(* PLC project VisuTest.project, CODESYS CODESYS V3.5 SP17 Patch 2 *)
(* stored: creationDateTime 2022-02-17T09:26:16.669529, modificationDateTime 2022-02-16T16:05:59.7420926, externalized true, stored C:\development\github\xml2ooxml\out\ex_contentHeader_12.xml *)

TYPE DUT : STRUCT

END_STRUCT;
END_TYPE

PROGRAM PLC_PRG
  VAR
    Counter : INT;
    ButtonPressed : BOOL;
    ButtonTrigger : R_TRIG;
    ResetPressed : BOOL;
    ResetTrigger : R_TRIG;
  END_VAR

                    ButtonTrigger(CLK:= ButtonPressed, Q=> );
IF (ButtonTrigger.Q) THEN
	Counter := Counter + 1;
END_IF

ResetTrigger(CLK:= ResetPressed, Q=> );
IF (ResetTrigger.Q) THEN
	Counter := 0;
END_IF
                  
END_PROGRAM

FUNCTION_BLOCK POU
  VAR
    x : INT;
  END_VAR

                    x := x + 2;
                  
END_FUNCTION_BLOCK

CONFIGURATION Device
  RESOURCE Application ON PLC
    TASK MainTask(INTERVAL := T#20ms, PRIORITY := 1);
    TASK VISU_TASK(INTERVAL := T#100ms, PRIORITY := 31);
    TASK Task(INTERVAL := T#20ms, PRIORITY := 1);
    PROGRAM PLC_PRG WITH MainTask : PLC_PRG;
    PROGRAM VisuElems.Visu_Prg WITH VISU_TASK : VisuElems.Visu_Prg;
  END_RESOURCE
END_CONFIGURATION
